FUNCTION_BLOCK PUBLIC PAEActuatorBase EXTENDS PAEControlModuleBase
VAR_INPUT
END_VAR
VAR_OUTPUT
END_VAR
VAR
END_VAR

METHOD PROTECTED GoToBasicPosition
VAR_INPUT
END_VAR
END_METHOD

METHOD PUBLIC IsEnabledSwitchToMaintenance : BOOL
VAR_INPUT
END_VAR
END_METHOD

METHOD PUBLIC SwitchToMaintenance
VAR_INPUT
END_VAR
END_METHOD

END_FUNCTION_BLOCK

(* stored: Version 1.1.0.1, ProductVersion 3.1.4020.12
   POU PAEActuatorBase: Id {1bec4bfa-032c-4c9e-a650-6604cbef6856}, SpecialFunc None
   Method GoToBasicPosition: Id {0ff620b3-085e-45af-8a6d-201bced75125}
   Method IsEnabledSwitchToMaintenance: Id {c4de3c36-74cf-48dc-b4e4-c1bcbd1090a0}
   Method SwitchToMaintenance: Id {f0bdd76c-5b0d-4b57-8229-0de5e68327d6} *)
